METHOD METH_RecipeFileInit : BOOL
VAR_INPUT
END_VAR
aRecipeParamsVariables[0]  :=  'stUBL.nRecipeIndexShow.diValue := '																				;   
aRecipeParamsVariables[1]  :=  'stUBL.iPackageCapTypeShow.diValue := '																	;       
aRecipeParamsVariables[2]  :=  'stUBL.iPackageCapDiameterShow.diValue := '																	;       
aRecipeParamsVariables[3]  :=  'stUBL.bExEnableShow.bValue := '																			;        
aRecipeParamsVariables[4]  :=  'stUBL.bBottleFeederEnableShow.bValue := '																;     
aRecipeParamsVariables[5]  :=  'stUBL.iBottleFeederTurntableVelocitySVShow.diValue := '																;        
aRecipeParamsVariables[6]  :=  'stUBL.iBottleFeederBottleSensorDelayShow.diValue := '																	;             
aRecipeParamsVariables[7]  :=  'stUBL.iBottleFeederFormGateDelayShow.diValue := '																	;             
aRecipeParamsVariables[8]  :=  'stUBL.iBottleFeederAllowFormDelayShow.diValue := '																	;               
aRecipeParamsVariables[9]  :=  'stUBL.bPucksInserterEnableShow.bValue := '															;
aRecipeParamsVariables[10] := 'stUBL.iPucksInserterTurntableVelocitySVShow.diValue := '															;    
aRecipeParamsVariables[11] := 'stUBL.iPucksInserterConveyorVelocitySVShow.diValue := '															;		
aRecipeParamsVariables[12] := 'stUBL.iPucksInserterBottleSensorDelayShow.diValue := '															;	
aRecipeParamsVariables[13] := 'stUBL.iPucksInserterFormGateDelayShow.diValue := '														;	
aRecipeParamsVariables[14] := 'stUBL.iPucksInserterAllowFormDelayShow.diValue := '														;	
aRecipeParamsVariables[15] := 'stUBL.lrPucksInserterWheelOffsetShow.lrValue := '															;
aRecipeParamsVariables[16] := 'stUBL.lrPucksInserterWheelAccelerationShow.lrValue := '																;			
aRecipeParamsVariables[17] := 'stUBL.lrPucksInserterWheelVelocityShow.lrValue := '																;			
aRecipeParamsVariables[18] := 'stUBL.lrPucksInserterHammerHeightSVShow.lrValue := '																;			
aRecipeParamsVariables[19] := 'stUBL.bGateBeforeDispencersEnableShow.bValue := '																;			
aRecipeParamsVariables[20] := 'stUBL.nGateBeforeDispencersTimeFormInsertingShow.lrValue := '																;			
aRecipeParamsVariables[21] := 'stUBL.bGateAfterWeightEnableShow.bValue := '																;			
aRecipeParamsVariables[22] := 'stUBL.nGateAfterWeightTimeFormInsertingShow.lrValue := '															;
aRecipeParamsVariables[23] := 'stUBL.bGateRobotEnableShow.bValue := '		      																	  ;
aRecipeParamsVariables[24] := 'stUBL.nGateRobotTimeFormInsertingShow.lrValue := '															            ;
aRecipeParamsVariables[25] := 'stUBL.bFormsDragingLeftEnableShow.bValue := '	        												    ;
aRecipeParamsVariables[26] := 'stUBL.lrFormsDragingLeftVelocityShow.lrValue := '	        												    ;
aRecipeParamsVariables[27] := 'stUBL.lrFormsDragingLeftAccelerationShow.lrValue := '														   	        ;
aRecipeParamsVariables[28] := 'stUBL.lrFormsDragingLeftDecelerationShow.lrValue := '	   													            ;
aRecipeParamsVariables[29] := 'stUBL.bFormsDragingRightEnableShow.bValue := '															            ;
aRecipeParamsVariables[30] := 'stUBL.lrFormsDragingRightVelocityShow.lrValue := '															            ;
aRecipeParamsVariables[31] := 'stUBL.lrFormsDragingRightAccelerationShow.lrValue := '															            ;
aRecipeParamsVariables[32] := 'stUBL.lrFormsDragingRightDecelerationShow.lrValue := '															            ;
aRecipeParamsVariables[33] := 'stUBL.bDosingTwoPhasesShow.bValue := '			        												    ;
aRecipeParamsVariables[34] := 'stUBL.lrDispencersLifterReadyPositionShow.lrValue := '															            ;
aRecipeParamsVariables[35] := 'stUBL.uiDispencerStartDosingDelayShow.udiValue := '														        ;
aRecipeParamsVariables[36] := 'stUBL.bDispencer1EnableShow.bValue := '	          																									  ;
aRecipeParamsVariables[37] := 'stUBL.bDispencer2EnableShow.bValue := '			  																									      ;
aRecipeParamsVariables[38] := 'stUBL.bDispencer3EnableShow.bValue := '	          													  ;
aRecipeParamsVariables[39] := 'stUBL.bDispencer4EnableShow.bValue := '				       									     ;
aRecipeParamsVariables[40] := 'stUBL.lrDispencer1DoseVolumeShow.lrValue := '				   									         ;
aRecipeParamsVariables[41] := 'stUBL.lrDispencer1Phase1VolumeShow.lrValue:= '	           									             ;
aRecipeParamsVariables[42] := 'stUBL.lrDispencer1Phase2VolumeShow.lrValue := '		       									         ;
aRecipeParamsVariables[43] := 'stUBL.lrDispencer1Phase1VelocityShow.lrValue := '		       									         ;
aRecipeParamsVariables[44] := 'stUBL.lrDispencer1Phase2VelocityShow.lrValue := '															;
aRecipeParamsVariables[45] := 'stUBL.lrDispencer1Phase3VelocityShow.lrValue := '			   									             ;
aRecipeParamsVariables[46] := 'stUBL.lrDispencer1SuckVelocityShow.lrValue := '			   									             ;
aRecipeParamsVariables[47] := 'stUBL.lrDispencer1Phase1AccelerationShow.lrValue := '												                ;
aRecipeParamsVariables[48] := 'stUBL.lrDispencer1Phase2AccelerationShow.lrValue := '		   									             ;
aRecipeParamsVariables[49] := 'stUBL.lrDispencer1Phase3AccelerationShow.lrValue := '		   									             ;
aRecipeParamsVariables[50] := 'stUBL.lrDispencer1SuckAccelerationShow.lrValue := '		   									             ;
aRecipeParamsVariables[51] := 'stUBL.lrDispencer1Phase1DecelerationShow.lrValue := '	       									         ;
aRecipeParamsVariables[52] := 'stUBL.lrDispencer1Phase2DecelerationShow.lrValue := '												                ;
aRecipeParamsVariables[53] := 'stUBL.lrDispencer1Phase3DecelerationShow.lrValue := '		   									                 ;
aRecipeParamsVariables[54] := 'stUBL.udiDispencer1DosingDoneDelayTimeShow.udiValue := '											                    ;
aRecipeParamsVariables[55] := 'stUBL.lrDispencer1SuckValveOpenVolumeShow.lrValue := '											                ;
aRecipeParamsVariables[56] := 'stUBL.lrDispencer1SuckValveOpenTimeDelayShow.lrValue := '											                ;
aRecipeParamsVariables[57] := 'stUBL.lrDispencer1SuckValveCloseVolumeShow.lrValue := '											                ;
aRecipeParamsVariables[58] := 'stUBL.lrDispencer1SuckValveCloseTimeDelayShow.lrValue := '										                    ;
aRecipeParamsVariables[59] := 'stUBL.lrDispencer1DoseValveOpenVolumeShow.lrValue := '	   									             ;
aRecipeParamsVariables[60] := 'stUBL.lrDispencer1DoseValveOpenTimeAccShow.lrValue := '      									               ;
aRecipeParamsVariables[61] := 'stUBL.lrDispencer1DoseValveCloseVolumeShow.lrValue := '      									               ;
aRecipeParamsVariables[62] := 'stUBL.lrDispencer1DoseValveCloseTimeDecShow.lrValue := '												                ;
aRecipeParamsVariables[63] := 'stUBL.lrDispencer1DoseSuckingVolumeShow.lrValue := '												                ;
aRecipeParamsVariables[64] := 'stUBL.lrDispencer1DoseSuckingTimeDelayShow.lrValue := '												                ;
aRecipeParamsVariables[65] := 'stUBL.bDispencer1DoseSuckingShow.bValue := '			       									         ;
aRecipeParamsVariables[66] := 'stUBL.bDispencer1LiftSynchroPh1Show.bValue := '																;
aRecipeParamsVariables[67] := 'stUBL.bDispencer1LiftSynchroPh2Show.bValue := '			   									             ;
aRecipeParamsVariables[68] := 'stUBL.bDispencer1LiftSynchroPh3Show.bValue := '		       									         ;
aRecipeParamsVariables[69] := 'stUBL.lrDispencer1LifterStartDosePositionShow.lrValue := '								                ;
aRecipeParamsVariables[70] := 'stUBL.lrDispencer1LifterStopDosePositionShow.lrValue := '										                ;
aRecipeParamsVariables[71] := 'stUBL.lrDispencer1LifterVelocityShow.lrValue := '	            							    ;
aRecipeParamsVariables[72] := 'stUBL.lrDispencer1LifterAccelerationShow.lrValue := '	        							        ;
aRecipeParamsVariables[73] := 'stUBL.lrDispencer1LifterDecelerationShow.lrValue := '		    							            ;
aRecipeParamsVariables[74] := 'stUBL.lrDispencer2DoseVolumeShow.lrValue := '		            							    ;
aRecipeParamsVariables[75] := 'stUBL.lrDispencer2Phase1VolumeShow.lrValue := '			    							            ;
aRecipeParamsVariables[76] := 'stUBL.lrDispencer2Phase2VolumeShow.lrValue := '			    							            ;
aRecipeParamsVariables[77] := 'stUBL.lrDispencer2Phase1VelocityShow.lrValue := '			    							            ;
aRecipeParamsVariables[78] := 'stUBL.lrDispencer2Phase2VelocityShow.lrValue := '			    							            ;
aRecipeParamsVariables[79] := 'stUBL.lrDispencer2Phase3VelocityShow.lrValue := '			    							            ;
aRecipeParamsVariables[80] := 'stUBL.lrDispencer2SuckVelocityShow.lrValue := '			    							            ;
aRecipeParamsVariables[81] := 'stUBL.lrDispencer2Phase1AccelerationShow.lrValue := '	        							        ;
aRecipeParamsVariables[82] := 'stUBL.lrDispencer2Phase2AccelerationShow.lrValue := '	        							        ;
aRecipeParamsVariables[83] := 'stUBL.lrDispencer2Phase3AccelerationShow.lrValue := '		    							            ;
aRecipeParamsVariables[84] := 'stUBL.lrDispencer2SuckAccelerationShow.lrValue := '	        							        ;
aRecipeParamsVariables[85] := 'stUBL.lrDispencer2Phase1DecelerationShow.lrValue := '											                ;
aRecipeParamsVariables[86] := 'stUBL.lrDispencer2Phase2DecelerationShow.lrValue := '											                ;
aRecipeParamsVariables[87] := 'stUBL.lrDispencer2Phase3DecelerationShow.lrValue := '											                ;
aRecipeParamsVariables[88] := 'stUBL.udiDispencer2DosingDoneDelayTimeShow.udiValue := '													;
aRecipeParamsVariables[89] := 'stUBL.lrDispencer2SuckValveOpenVolumeShow.lrValue := '									                ;
aRecipeParamsVariables[90] := 'stUBL.lrDispencer2SuckValveOpenTimeDelayShow.lrValue := '											                ;
aRecipeParamsVariables[91] := 'stUBL.lrDispencer2SuckValveCloseVolumeShow.lrValue := '											                ;
aRecipeParamsVariables[92] := 'stUBL.lrDispencer2SuckValveCloseTimeDelayShow.lrValue := '											                ;
aRecipeParamsVariables[93] := 'stUBL.lrDispencer2DoseValveOpenVolumeShow.lrValue := '										                ;
aRecipeParamsVariables[94] := 'stUBL.lrDispencer2DoseValveOpenTimeAccShow.lrValue := '									                    ;
aRecipeParamsVariables[95] := 'stUBL.lrDispencer2DoseValveCloseVolumeShow.lrValue := '									                    ;
aRecipeParamsVariables[96] := 'stUBL.lrDispencer2DoseValveCloseTimeDecShow.lrValue := '										                    ;
aRecipeParamsVariables[97] := 'stUBL.lrDispencer2DoseSuckingVolumeShow.lrValue := '		    							                    ;
aRecipeParamsVariables[98] := 'stUBL.lrDispencer2DoseSuckingTimeDelayShow.lrValue := '									                        ;
aRecipeParamsVariables[99] := 'stUBL.bDispencer2DoseSuckingShow.bValue := '		            							        ;
aRecipeParamsVariables[100]:= 'stUBL.bDispencer2LiftSynchroPh1Show.bValue := '		        							            ;
aRecipeParamsVariables[101]:= 'stUBL.bDispencer2LiftSynchroPh2Show.bValue := '		        							            ;
aRecipeParamsVariables[102]:= 'stUBL.bDispencer2LiftSynchroPh3Show.bValue := '		        							        ;
aRecipeParamsVariables[103]:= 'stUBL.lrDispencer2LifterStartDosePositionShow.lrValue := '								  	                    ;
aRecipeParamsVariables[104]:= 'stUBL.lrDispencer2LifterStopDosePositionShow.lrValue := '								  	            ;
aRecipeParamsVariables[105]:= 'stUBL.lrDispencer2LifterVelocityShow.lrValue := '	        							            ;
aRecipeParamsVariables[106]:= 'stUBL.lrDispencer2LifterAccelerationShow.lrValue := '									                ;
aRecipeParamsVariables[107]:= 'stUBL.lrDispencer2LifterDecelerationShow.lrValue := '	    							                ;
aRecipeParamsVariables[108]:= 'stUBL.bDispencersCatchEnableShow.bValue := '	            							    ;
aRecipeParamsVariables[109]:= 'stUBL.bDispencersCatchMaxPressureShow.bValue := '           							         ;
aRecipeParamsVariables[110]:= 'stUBL.lrDispencersCatchHeightSVShow.lrValue := '														;
aRecipeParamsVariables[111]:= 'stUBL.lrDispencersCatch1ClosedValueShow.lrValue := '         							       ;
aRecipeParamsVariables[112]:= 'stUBL.lrDispencersCatch1OpenValueShow.lrValue := '           							   ;
aRecipeParamsVariables[113]:= 'stUBL.lrDispencersCatch2ClosedValueShow.lrValue := '         							         ;
aRecipeParamsVariables[114]:= 'stUBL.lrDispencersCatch2OpenValueShow.lrValue := '		    							            ;
aRecipeParamsVariables[115]:= 'stUBL.lrDispencersCatch3ClosedValueShow.lrValue := '         							       ;
aRecipeParamsVariables[116]:= 'stUBL.lrDispencersCatch3OpenValueShow.lrValue := '           							        ;
aRecipeParamsVariables[117]:= 'stUBL.lrDispencersCatch4ClosedValueShow.lrValue := '         							        ;
aRecipeParamsVariables[118]:= 'stUBL.lrDispencersCatch4OpenValueShow.lrValue := '										;								
aRecipeParamsVariables[119]:= 'stUBL.lrDispencersCatchToleranceShow.lrValue := '	        							;
aRecipeParamsVariables[120]:= 'stUBL.bTank1MixerEnableShow.bValue := '    												 ;
aRecipeParamsVariables[121]:= 'stUBL.bTankHeatingEnableShow.bValue := '   												                ;
aRecipeParamsVariables[122]:= 'stUBL.iTankHeatingTempSVShow.diValue := '   												      ;
aRecipeParamsVariables[123]:= 'stUBL.bTank1PressureEnableShow.bValue := ' 														;
aRecipeParamsVariables[124]:= 'stUBL.bTank1SupplyPumpEnableShow.bValue := '	                                           ;
aRecipeParamsVariables[125]:= 'stUBL.bTank2SupplyPumpEnableShow.bValue := '	                                           ;
aRecipeParamsVariables[126]:= 'stUBL.uTank1LevelSetpointShow.udiValue := '	                                           ;
aRecipeParamsVariables[127]:= 'stUBL.uTank2LevelSetpointShow.udiValue := '	                                           ;
aRecipeParamsVariables[128]:= 'stUBL.bTank1LevelSignalInvertShow.bValue := '	                                           ;
aRecipeParamsVariables[129]:= 'stUBL.bTank2LevelSignalInvertShow.bValue := '	                                           ;
aRecipeParamsVariables[130]:= 'stUBL.bWeight1EnableShow.bValue := '	                                           ;
aRecipeParamsVariables[131]:= 'stUBL.lrWeightMassSVShow.lrValue := '	                                           ;
aRecipeParamsVariables[132]:= 'stUBL.iWeight1ActuatorUpDelayShow.diValue := '											  ;	
aRecipeParamsVariables[133]:= 'stUBL.iWeight2ActuatorUpDelayShow.diValue := '	                                           ;
aRecipeParamsVariables[134]:= 'stUBL.iWeight3ActuatorUpDelayShow.diValue := '	                                           ;
aRecipeParamsVariables[135]:= 'stUBL.iWeight4ActuatorUpDelayShow.diValue := '	                                           ;
aRecipeParamsVariables[136]:= 'stUBL.iWeight5ActuatorUpDelayShow.diValue := '	                                           ;
aRecipeParamsVariables[137]:= 'stUBL.iWeight6ActuatorUpDelayShow.diValue := '	                                           ;
aRecipeParamsVariables[138]:= 'stUBL.lrFormWeightShow.lrValue := '	                                           ;
aRecipeParamsVariables[139]:= 'stUBL.lrMass1DensityShow.lrValue := '	                                           ;
aRecipeParamsVariables[140]:= 'stUBL.lrMass2DensityShow.lrValue := '	                                           ;
aRecipeParamsVariables[141]:= 'stUBL.lrCupWeightShow.lrValue := '	                                           ;
aRecipeParamsVariables[142]:= 'stUBL.lrWholePackageWeightShow.lrValue := '	                                           ;
aRecipeParamsVariables[143]:= 'stUBL.lrWeight1MeasurmentCorrectionShow.lrValue := '	                                           ;
aRecipeParamsVariables[144]:= 'stUBL.bDispencer1WeightCorrectionEnableShow.bValue := '	                                           ;
aRecipeParamsVariables[145]:= 'stUBL.bDispencer2WeightCorrectionEnableShow.bValue := '	                                           ;
aRecipeParamsVariables[146]:= 'stUBL.bDispencer3WeightCorrectionEnableShow.bValue := '	                                           ;
aRecipeParamsVariables[147]:= 'stUBL.bDispencer4WeightCorrectionEnableShow.bValue := '	                                           ;
aRecipeParamsVariables[148]:= 'stUBL.lrWeightUpperToleranceShow.lrValue := '	                                           ;
aRecipeParamsVariables[149]:= 'stUBL.lrWeightLowerToleranceShow.lrValue := '	                                           ;
aRecipeParamsVariables[150]:= 'stUBL.iWeightCorrectionNumberOfSamplesShow.diValue := '	                                           ;
aRecipeParamsVariables[151]:= 'stUBL.bLidFeederEnableShow.bValue := '	                                           ;
aRecipeParamsVariables[152]:= 'stUBL.bLidFeederHeaterEnableShow.bValue := '	                                           ;
aRecipeParamsVariables[153]:= 'stUBL.lrLidFeederHeightPosSVShow.lrValue := '	                                           ;
aRecipeParamsVariables[154]:= 'stUBL.iLidFeederHeatingTimeShow.diValue := '	                                           ;
aRecipeParamsVariables[155]:= 'stUBL.iLidFeederTempHisteresisShow.diValue := '	                                           ;
aRecipeParamsVariables[156]:= 'stUBL.iLidFeeder1TempSVShow.diValue := '	                                           ;
aRecipeParamsVariables[157]:= 'stUBL.iLidFeeder2TempSVShow.diValue := '	                                           ;
aRecipeParamsVariables[158]:= 'stUBL.bLidFeederDragingStationEnableShow.bValue := '	                                           ;
aRecipeParamsVariables[159]:= 'stUBL.lrLidFeederDragingStationVelocityShow.lrValue := '	                                           ;
aRecipeParamsVariables[160]:= 'stUBL.lrLidFeederDragingStationAccelerationShow.lrValue := '	                                           ;
aRecipeParamsVariables[161]:= 'stUBL.lrLidFeederDragingStationDecelerationShow.lrValue := '	                                           ;
aRecipeParamsVariables[162]:= 'stUBL.bLidPuttedCheckEnableShow.bValue := '	                                           ;
aRecipeParamsVariables[163]:= 'stUBL.lrLidPuttedCheckHeightSVShow.lrValue := '	                                           ;
aRecipeParamsVariables[164]:= 'stUBL.lrLidPuttedCheckPositionShow.lrValue := '	                                           ;
aRecipeParamsVariables[165]:= 'stUBL.lrLidPuttedCheckAreaShow.lrValue := '	                                           ;
aRecipeParamsVariables[166]:= 'stUBL.iLidPuttedCheckProgramShow.diValue := '	                                           ;
aRecipeParamsVariables[167]:= 'stUBL.bLidSealerEnableSho.bValuew := '	                                           ;
aRecipeParamsVariables[168]:= 'stUBL.bLidSealerHeaterEnableShow.bValue := '	                                           ;
aRecipeParamsVariables[169]:= 'stUBL.iLidSealerHeatingTimeShow.diValue := '	                                           ;
aRecipeParamsVariables[170]:= 'stUBL.lrLidSealerPressureShow.lrValue := '	                                           ;
aRecipeParamsVariables[171]:= 'stUBL.lrLidSealerHeightPosSVShow.lrValue := '	                                           ;
aRecipeParamsVariables[172]:= 'stUBL.iLidSealerTempHisteresisShow.diValue := '	                                           ;
aRecipeParamsVariables[173]:= 'stUBL.iLidSealer1TempSVShow.diValue := '	                                           ;
aRecipeParamsVariables[174]:= 'stUBL.iLidSealer2TempSVShow.diValue := '	                                           ;
aRecipeParamsVariables[175]:= 'stUBL.bLidSealerDragingStationEnableShow.bValue := '	                                           ;
aRecipeParamsVariables[176]:= 'stUBL.lrLidSealerDragingStationVelocityShow.lrValue := '	                                           ;
aRecipeParamsVariables[177]:= 'stUBL.lrLidSealerDragingStationAccelerationShow.lrValue := '	                                           ;
aRecipeParamsVariables[178]:= 'stUBL.lrLidSealerDragingStationDecelerationShow.lrValue := '	                                           ;
aRecipeParamsVariables[179]:= 'stUBL.bCapFeederGateEnableShow.bValue := '	                                           ;
aRecipeParamsVariables[180]:= 'stUBL.iCapFeederGateBlockingTimeShow.diValue := '	                                           ;
aRecipeParamsVariables[181]:= 'stUBL.bCapFeederEnableShow.bValue := '	                                           ;
aRecipeParamsVariables[182]:= 'stUBL.lrCapFeederHeightPosSVShow.lrValue := '	                                           ;
aRecipeParamsVariables[183]:= 'stUBL.iCapFeederTimeDelayOnShow.diValue := '                                            ;
aRecipeParamsVariables[184]:= 'stUBL.iCapFeederTimeDelayOffShow.diValue := '                                            ;
aRecipeParamsVariables[185]:= 'stUBL.iCapFeederTimeToEmptySleeveErrorShow.diValue := '	                                           ;
aRecipeParamsVariables[186]:= 'stUBL.bCapSorterOnlyWeightOKEnableShow.bValue := '	                                           ;
aRecipeParamsVariables[187]:= 'stUBL.bCapSorterDragEnableShow.bValue := '	                                           ;
aRecipeParamsVariables[188]:= 'stUBL.lrCapSorterDragVelocityShow.lrValue := '	                                           ;
aRecipeParamsVariables[189]:= 'stUBL.lrCapSorterDragAccelerationShow.lrValue := '	                                           ;
aRecipeParamsVariables[190]:= 'stUBL.lrCapSorterDragDecelerationShow.lrValue := '	                                           ;
aRecipeParamsVariables[191]:= 'stUBL.bCapPuttedCheckEnableShow.bValue := '	                                           ;
aRecipeParamsVariables[192]:= 'stUBL.lrCapPuttedCheckHeightPosSVShow.lrValue := '	                                           ;
aRecipeParamsVariables[193]:= 'stUBL.bGripperScrewer1EnableShow.bValue := '	                                           ;
aRecipeParamsVariables[194]:= 'stUBL.lrGripperScrewingTightTorqueShow.lrValue := '	                                           ;
aRecipeParamsVariables[195]:= 'stUBL.bGripperScrewer2EnableShow.bValue := '	                                           ;
aRecipeParamsVariables[196]:= 'stUBL.lrGripperScrewing2TightTorqueShow.lrValue := '	                                           ;
aRecipeParamsVariables[197]:= 'stUBL.iGripperScrewer1ToolShow.diValue := '	                                           ;
aRecipeParamsVariables[198]:= 'stUBL.lrGripperScrewer1VelocityShow.lrValue := '	                                           ;
aRecipeParamsVariables[199]:= 'stUBL.nGripperScrewer1TightTimeShow.udiValue := '	                                           ;
aRecipeParamsVariables[200]:= 'stUBL.iGripperScrewer1StartDelayShow.diValue := '	                                           ;
aRecipeParamsVariables[201]:= 'stUBL.lrGripperScrewerReadyPositionShow.lrValue := '	                                           ;
aRecipeParamsVariables[202]:= 'stUBL.lrGripperScrewerPushingCapPositionShow.lrValue := '	                                           ;
aRecipeParamsVariables[203]:= 'stUBL.lrGripperScrewerScrewingCapPositionShow.lrValue := '	                                           ;
aRecipeParamsVariables[204]:= 'stUBL.lrGripperScrewerPressureShow.lrValue := '	                                           ;
aRecipeParamsVariables[205]:= 'stUBL.lrGripperScrewerCatchPressureShow.lrValue := '	                                           ;
aRecipeParamsVariables[206]:= 'stUBL.lrDispencerCatchPressureShow.lrValue := '	                                           ;
aRecipeParamsVariables[207]:= 'stUBL.lrGripperScrewerPressureExhaustLevelShow.lrValue := '	                                           ;
aRecipeParamsVariables[208]:= 'stUBL.lrGripperScrewerCatchPressureExhaustLevelShow.lrValue := '	                                           ;
aRecipeParamsVariables[209]:= 'stUBL.lrGripperScrewerTurnoversToFullScrewedShow.lrValue := '	                                           ;
aRecipeParamsVariables[210]:= 'stUBL.lrGripperScrewerThreadPitchShow.lrValue := '	                                           ;
aRecipeParamsVariables[211]:= 'stUBL.lrGripperScrewerThreadTimesShow.lrValue := '	                                           ;
aRecipeParamsVariables[212]:= 'stUBL.nGripperScrewerCatchHeightSVShow.udiValue := '	                           								                ;
aRecipeParamsVariables[213]:= 'stUBL.bGripperScrewer1FindScrewShow.bValue := '	                		            ;
aRecipeParamsVariables[214]:= 'stUBL.bGripperScrewer1Option4Show.bValue := '	                		            ;
aRecipeParamsVariables[215]:= 'stUBL.lrGripperScrewer1FindingScrewDegreeShow.lrValue := '	    		                        ;
aRecipeParamsVariables[216]:= 'stUBL.bGripperScrewer1Option1Show.bValue := '	                		            ;
aRecipeParamsVariables[217]:= 'stUBL.bGripperScrewer1Option2Show.bValue := '	                		            ;
aRecipeParamsVariables[218]:= 'stUBL.bGripperScrewer1Option3Show.bValue := '	                		            ;
aRecipeParamsVariables[219]:= 'stUBL.bGripperScrewer1Option5Show.bValue := '	                		            ;
aRecipeParamsVariables[220]:= 'stUBL.bGripperScrewer1Option6Show.bValue := '	                		            ;
aRecipeParamsVariables[221]:= 'stUBL.bGripperScrewer1Option7Show.bValue := '	                		            ;
aRecipeParamsVariables[222]:= 'stUBL.bBottleDragingStationEnableShow.bValue := '	            		                ;
aRecipeParamsVariables[223]:= 'stUBL.lrBottleDragingStationVelocityShow.lrValue := '	        		                    ;
aRecipeParamsVariables[224]:= 'stUBL.bCapCorrectCheckEnableShow.bValue := '	                    	            ;
aRecipeParamsVariables[225]:= 'stUBL.lrCapCorrectCheckHeightPosSVShow.lrValue := '	            		                ;
aRecipeParamsVariables[226]:= 'stUBL.bCapCorrectCheckCameraEnableShow.bValue := '	            		                ;
aRecipeParamsVariables[227]:= 'stUBL.iCapCorrectCheckCameraProgramShow.diValue := '	            		                ;
aRecipeParamsVariables[228]:= 'stUBL.bBottleTransferEnableShow.bValue		 := '	            		                ;
aRecipeParamsVariables[229]:= 'stUBL.nBottleTransferProgramShow.udiValue		 := '	        			                ;
aRecipeParamsVariables[230]:= 'stUBL.iBottleTransferPickOffsetXShow.diValue  := '	            		                ;
aRecipeParamsVariables[231]:= 'stUBL.iBottleTransferPickOffsetYShow.diValue  := '	            		                ;
aRecipeParamsVariables[232]:= 'stUBL.iBottleTransferPickOffsetZShow.diValue  := '	            		                ;
aRecipeParamsVariables[233]:= 'stUBL.iBottleTransferPick2OffsetXShow.diValue := '	            		                ;
aRecipeParamsVariables[234]:= 'stUBL.iBottleTransferPick2OffsetYShow.diValue := '	            		                ;
aRecipeParamsVariables[235]:= 'stUBL.iBottleTransferPick2OffsetZShow.diValue := '	            		                ;
aRecipeParamsVariables[236]:= 'stUBL.iBottleTransferPlace1OffsetXShow.diValue := '	            		                ;
aRecipeParamsVariables[237]:= 'stUBL.iBottleTransferPlace1OffsetYShow.diValue := '	            		                ;
aRecipeParamsVariables[238]:= 'stUBL.iBottleTransferPlace1OffsetZShow.diValue := '	            		                ;
aRecipeParamsVariables[239]:= 'stUBL.iBottleTransferPlace2OffsetXShow.diValue := '	            		                ;
aRecipeParamsVariables[240]:= 'stUBL.iBottleTransferPlace2OffsetYShow.diValue := '	            		                ;
aRecipeParamsVariables[241]:= 'stUBL.iBottleTransferPlace2OffsetZShow.diValue := '	            		                ;
aRecipeParamsVariables[242]:= 'stUBL.iBottleTransferSpeedShow.diValue := '	                    		        ;
aRecipeParamsVariables[243]:= 'stUBL.bBottleTransferInkJetEnableShow.bValue := '	            		                ;
aRecipeParamsVariables[244]:= 'stUBL.bBottleTransferPickOnlyOneShow.bValue := '	                	                ;
aRecipeParamsVariables[245]:= 'stUBL.bBottleTransferWeightEnableShow.bValue := '	            		  							              ;
aRecipeParamsVariables[246]:= 'stUBL.iBottleTransferWeightIntervalShow.diValue := '	            		              ;
aRecipeParamsVariables[247]:= 'stUBL.bBottleTransferRotateEnableShow.bValue := '	            		              ;
aRecipeParamsVariables[248]:= 'stUBL.bBadBottleConveyorEnableShow.bValue := '	                		          ;
aRecipeParamsVariables[249]:= 'stUBL.nBadBottleConveyorVelocitySVShow.udiValue := '	            		              ;
aRecipeParamsVariables[250]:= 'stUBL.bLabelMachineEnableShow.bValue := '	                    		      ;
aRecipeParamsVariables[251]:= 'stUBL.bExitTurnTable1EnableShow.bValue := '	                    		      ;
aRecipeParamsVariables[252]:= 'stUBL.bExitConveyorEnableShow.bValue := '	                    		      ;
aRecipeParamsVariables[253]:= 'stUBL.nExitConveyorVelocitySVShow.udiValue := '	                		          ;
aRecipeParamsVariables[254]:= 'stUBL.bFormTransportersEnableShow.bValue					 := '		                              ;
aRecipeParamsVariables[255]:= 'stUBL.nFormTransportersDispencerVelocitySVShow.udiValue	 := '	                 							                          ;
aRecipeParamsVariables[256]:= 'stUBL.nFormTransportersScrewerVelocitySVShow.udiValue		 := '	                 							                          ;
aRecipeParamsVariables[257]:= 'stUBL.nFormTransportersBeforeScrewerVelocitySVShow.udiValue := '	                 				                          ;
aRecipeParamsVariables[258]:= 'stUBL.nFormTransportersSlowerVelocitySVShow.udiValue		 := '	                 				                          ;
aRecipeParamsVariables[259]:= 'stUBL.bCircularInkjetEnableShow.bValue	 := '	                                 				          ;
aRecipeParamsVariables[260]:= 'stUBL.iCircularInkjetSpeedShow.diValue	 := '	                                 				          ;
aRecipeParamsVariables[261]:= 'stUBL.iCircularInkjetDelayShow.diValue	 := '	                                 				          ;
aRecipeParamsVariables[262]:= 'stUBL.iCircularInkjetHoldShow.diValue	 := '	                                 				          ;
aRecipeParamsVariables[263]:= 'stUCF.iCapSorterProductType.diValue := '	                                         								  ;
aRecipeParamsVariables[264]:= 'stUCF.uiCapSorterIndexShow.udiValue := '																						;
aRecipeParamsVariables[265]:= 'stUCF.bPresenceBottleEnableShow.bValue := '	                                     									                                ;
aRecipeParamsVariables[266]:= 'stUCF.bCapSorterTransporterEnableShow.bValue								 := '	  					     ;
aRecipeParamsVariables[267]:= 'stUCF.iCapSorterTransporterTankConveyorVelocityShow.diValue				 := '	    					   ;
aRecipeParamsVariables[268]:= 'stUCF.iCapSorterTransporterStartDelayTimeShow.diValue						 := '						  ;
aRecipeParamsVariables[269]:= 'stUCF.udiCapSorterTransporterTimeProductOnSensorBeforeBrushShow.udiValue	 := '										            ;
aRecipeParamsVariables[270]:= 'stUCF.iCapSorterTransporterEmptyingConveyorSpeedShow.diValue				 := '					            ;
aRecipeParamsVariables[271]:= 'stUCF.iCapSorterTransporterVolumeOfCapsShow.diValue						 := '					            ;
aRecipeParamsVariables[272]:= 'stUCF.bCapSorterWheelEnableShow.bValue							 := '	        				     ;
aRecipeParamsVariables[273]:= 'stUCF.lrCapSorterWheelMoveAccelerationEmptyTableShow.lrValue		 := '	        				   	 ;
aRecipeParamsVariables[274]:= 'stUCF.lrCapSorterWheelMoveDecelerationEmptyTableShow.lrValue		 := '	        				   	 ;
aRecipeParamsVariables[275]:= 'stUCF.lrCapSorterWheelMoveSpeedEmptyTableShow.lrValue				 := '	    				        ;
aRecipeParamsVariables[276]:= 'stUCF.lrCapSorterWheelMoveAngleEmptyTableShow.lrValue				 := '	    				        ;
aRecipeParamsVariables[277]:= 'stUCF.lrCapSorterWheelJerkAngleEmptyTableShow.lrValue				 := '	    				        ;
aRecipeParamsVariables[278]:= 'stUCF.iCapSorterWheelWaitingAfterRotationEmptyTableShow.diValue := '	            				    ;
aRecipeParamsVariables[279]:= 'stUCF.lrCapSorterWheelMoveAccelerationFullTableShow.lrValue	 := '	            				    ;
aRecipeParamsVariables[280]:= 'stUCF.lrCapSorterWheelMoveDecelerationFullTableShow.lrValue	 := '	            				   ;
aRecipeParamsVariables[281]:= 'stUCF.lrCapSorterWheelMoveSpeedFullTableShow.lrValue			 := '	            				    ;
aRecipeParamsVariables[282]:= 'stUCF.lrCapSorterWheelMoveAngleFullyTableShow.lrValue			 := '           				   ;
aRecipeParamsVariables[283]:= 'stUCF.lrCapSorterWheelJerkAngleFullTableShow.lrValue			 := '               				   ;
aRecipeParamsVariables[284]:= 'stUCF.iCapSorterWheelWaitingAfterRotationFullTableShow.diValue := '	           											    ;
aRecipeParamsVariables[285]:= 'stUCF.lrCapSorterWheelMoveAccelerationHalfFullTableShow.lrValue	 := '	       											     ;
aRecipeParamsVariables[286]:= 'stUCF.lrCapSorterWheelMoveDecelerationHalfFullTableShow.lrValue	 := '	       				     ;
aRecipeParamsVariables[287]:= 'stUCF.lrCapSorterWheelMoveSpeedHalfFullTableShow.lrValue			 := '	       				     ;
aRecipeParamsVariables[288]:= 'stUCF.lrCapSorterWheelMoveAngleHalfFullyTableShow.lrValue			 := '	   				         ;
aRecipeParamsVariables[289]:= 'stUCF.lrCapSorterWheelJerkAngleHalfFullTableShow.lrValue			 := '	       				     ;
aRecipeParamsVariables[290]:= 'stUCF.iCapSorterWheelWaitingAfterRotationHalfFullTableShow.diValue := '	       				     ;
aRecipeParamsVariables[291]:= 'stUCF.bCapSorterCameraEnableShow.bValue := '     ;                             				
aRecipeParamsVariables[292]:= 'stUCF.bCapSorterRobotEnableShow.bValue := '	 ;                                 				
aRecipeParamsVariables[293]:= 'stUCF.lrCapSorterRobotPlace1PositionXShow.lrValue			 := '									     ;
aRecipeParamsVariables[294]:= 'stUCF.lrCapSorterRobotPlace1PositionYShow.lrValue			 := '									     ;
aRecipeParamsVariables[295]:= 'stUCF.lrCapSorterRobotPlace1PositionZShow.lrValue			 := '									     ;
aRecipeParamsVariables[296]:= 'stUCF.lrCapSorterRobotPlace1PositionCShow.lrValue			 := '									     ;
aRecipeParamsVariables[297]:= 'stUCF.iCapSorterRobotPickElevationShow.diValue			 := '	    								 ;
aRecipeParamsVariables[298]:= 'stUCF.iCapSorterRobotPickTimeShow.diValue					 := '									     ;
aRecipeParamsVariables[299]:= 'stUCF.iCapSorterRobotVacuumActivationShow.diValue			 := '									     ;
aRecipeParamsVariables[300]:= 'stUCF.iCapSorterRobotVacuumOffShow.diValue				 := '	    								 ;
aRecipeParamsVariables[301]:= 'stUCF.iCapSorterRobotPlaceTimeShow.diValue				 := '	    								 ;
aRecipeParamsVariables[302]:= 'stUCF.iCapSorterRobotTCP_PlaceOffsetShow.diValue			 := '	    								 ;
aRecipeParamsVariables[303]:= 'stUCF.iCapSorterRobotAccelerationDecelerationShow.diValue	 := '									     ;
aRecipeParamsVariables[304]:= 'stUCF.iCapSorterRobotGripperWatchdogShow.diValue			 := '	    								 ;
aRecipeParamsVariables[305]:= 'stUCF.iCapSorterRobotParalaxCorrectionShow.diValue		 := '	    								 ;
aRecipeParamsVariables[306]:= 'stUCF.iCapSorterRobotNumberToolShow.diValue	 := '	 													 ;
aRecipeParamsVariables[307]:= 'stUCF.iCapSorterRobotPickPositionZShow.diValue := '	 													 ;
aRecipeParamsVariables[308]:= 'stUCF.iCapSorterRobotTCP_Lenght.diValue		 := '	 																			 ;
aRecipeParamsVariables[309]:= 'stUCF.iCapSorterRobotProductDiametr.diValue	 := '	 												 ;
aRecipeParamsVariables[310]:= 'stUCF.bCapSorterIntermediateTransporterEnableShow.bValue					 := '				     ;
aRecipeParamsVariables[311]:= 'stUCF.iCapSorterIntermediateTransporterAutoSpeedShow.diValue				 := '	    			 ;
aRecipeParamsVariables[312]:= 'stUCF.iCapSorterIntermediateTransporterManualSpeedShow.diValue			 := '	    			 ;
aRecipeParamsVariables[313]:= 'stUCF.iCapSorterIntermediateTransporterEmptyingSpeedShow.diValue			 := '	    			 ;
aRecipeParamsVariables[314]:= 'stUCF.iCapSorterIntermediateTransporterDelayCountTimeShow.diValue			 := '				     ;
aRecipeParamsVariables[315]:= 'stUCF.iCapSorterIntermediateTransporterReverseTimeShow.diValue			 := '	    			 ;
aRecipeParamsVariables[316]:= 'stUCF.udiCapSorterIntermediateTransporterTimeProductOnSensorShow.udiValue	 := '					 ;
aRecipeParamsVariables[317]:= 'stUCF.lrCapSorterIntermediateTransporterWheelAngleShow.lrValue			 := '	    			 ;
aRecipeParamsVariables[318]:= 'stUCF.bCapSorterIntermediateBrushEnableShow.bValue			 := '	  												      ;
aRecipeParamsVariables[319]:= 'stUCF.iCapSorterIntermediateBrushAutoSpeedShow.diValue		 := '	  												      ;
aRecipeParamsVariables[320]:= 'stUCF.iCapSorterIntermediateBrushManualSpeedShow.diValue		 := '	  						      ;
aRecipeParamsVariables[321]:= 'stUCF.iCapSorterIntermediateBrushEmptyingSpeedShow.diValue	 := '	  						      ;
aRecipeParamsVariables[322]:= 'stUCF.lrCapSorterIntermediateBrushPositionHeightSVShow.lrValue := '    						    ;
aRecipeParamsVariables[323]:= 'stUCF.bCapSorterBrush1OnWheelEnableShow.bValue			 := '      														  ;
aRecipeParamsVariables[324]:= 'stUCF.iCapSorterBrush1OnWheelAutoSpeedShow.diValue		 := '      					  ;
aRecipeParamsVariables[325]:= 'stUCF.iCapSorterBrush1OnWheelManualSpeedShow.diValue		 := '      					  ;
aRecipeParamsVariables[326]:= 'stUCF.iCapSorterBrush1OnWheelEmptyingSpeedShow.diValue	 := '      					  ;
aRecipeParamsVariables[327]:= 'stUCF.lrCapSorterBrush1OnWheelPositionHeightSVShow.lrValue := '     					   ;
aRecipeParamsVariables[328]:= 'stUCF.bCapSorterBrush2OnWheelEnableShow.bValue			 := '      					  ;
aRecipeParamsVariables[329]:= 'stUCF.iCapSorterBrush2OnWheelAutoSpeedShow.diValue		 := '      					  ;
aRecipeParamsVariables[330]:= 'stUCF.iCapSorterBrush2OnWheelManualSpeedShow.diValue		 := '      					  ;
aRecipeParamsVariables[331]:= 'stUCF.iCapSorterBrush2OnWheelEmptyingSpeedShow.diValue	 := '      					  ;
aRecipeParamsVariables[332]:= 'stUCF.lrCapSorterBrush2OnWheelPositionHeightSVShow.lrValue := '     					   ;
aRecipeParamsVariables[333]:= 'stUCF.bCapSorterFeederEnableShow.bValue					 := '      					  ;
aRecipeParamsVariables[334]:= 'stUCF.bCapSorterFeederEnableTubeError.bValue				 := '  						  ;
aRecipeParamsVariables[335]:= 'stUCF.lrCapSorterFeederMover1InputPositionShow.lrValue	 := '      					  ;
aRecipeParamsVariables[336]:= 'stUCF.lrCapSorterFeederMover2InputPositionShow.lrValue	 := '      					  ;
aRecipeParamsVariables[337]:= 'stUCF.lrCapSorterFeederMover1OutputPositionShow.lrValue	 := '      					  ;
aRecipeParamsVariables[338]:= 'stUCF.lrCapSorterFeederMover2OutputPositionShow.lrValue	 := '      					  ;
aRecipeParamsVariables[339]:= 'stUCF.lrCapSorterFeederSlotDistanceShow.lrValue			 := '      					  ;
aRecipeParamsVariables[340]:= 'stUCF.lrCapSorterFeederMoverSpeedShow.lrValue				 := '  					      ;
aRecipeParamsVariables[341]:= 'stUCF.lrCapSorterFeederMoverAccelerationShow.lrValue		 := '      					  ;
aRecipeParamsVariables[342]:= 'stUCF.lrCapSorterFeederMoveJerkShow.lrValue				 := '      					  ;
aRecipeParamsVariables[343]:= 'stUCF.bCapSorterPreScrewerEnableShow.bValue			 := '          					    ;
aRecipeParamsVariables[344]:= 'stUCF.bCapSorterPreScrewerPicker1EnableShow.bValue := '            					  ;
aRecipeParamsVariables[345]:= 'stUCF.bCapSorterPreScrewerPicker2EnableShow.bValue := '            					  ;
aRecipeParamsVariables[346]:= 'stUCF.bCapSorterPreScrewerPicker3EnableShow.bValue := '           													   ;
aRecipeParamsVariables[347]:= 'stUCF.bCapSorterPreScrewerPicker4EnableShow.bValue := '           																   ;
aRecipeParamsVariables[348]:= 'stUCF.lrCapSorterPreScrewerPickZPositionShow.lrValue					 := '       																 ;
aRecipeParamsVariables[349]:= 'stUCF.lrCapSorterPreScrewerCatcherReleseShow.lrValue					 := '       																 ;
aRecipeParamsVariables[350]:= 'stUCF.lrCapSorterPreScrewerCapCatcherZPositionShow.lrValue			 := '       																 ;
aRecipeParamsVariables[351]:= 'stUCF.lrCapSorterPreScrewerTopZPositionShow.lrValue					 := '       																 ;
aRecipeParamsVariables[352]:= 'stUCF.lrCapSorterPreScrewerCartesianCatchZPositionShow.lrValue		 := '       																 ;
aRecipeParamsVariables[353]:= 'stUCF.lrCapSorterPreScrewerStrawCatcherZPositionShow.lrValue			 := '       																 ;
aRecipeParamsVariables[354]:= 'stUCF.LrCapSorterPreScrewerCheckStrawCatcherActuatorZPosition.lrValue	 := '   																     ;
aRecipeParamsVariables[355]:= 'stUCF.lrCapSorterPreScrewerScrewerStartZPositionShow.lrValue			 := '       																 ;
aRecipeParamsVariables[356]:= 'stUCF.lrCapSorterPreScrewerGripperOpenPositionShow.lrValue			 := '       																 ;
aRecipeParamsVariables[357]:= 'stUCF.lrCapSorterPreScrewerPlaceZPositionShow.lrValue					 := '   																     ;
aRecipeParamsVariables[358]:= 'stUCF.lrCapSorterPreScrewerBendingDistanceShow.lrValue := '            ;
aRecipeParamsVariables[359]:= 'stUCF.lrCapSorterPreScrewerStrawInsertDistance.lrValue := '            ;
aRecipeParamsVariables[360]:= 'stUCF.lrCapSorterPreScrewerPickXMover1PositionShow.lrValue := '            ;
aRecipeParamsVariables[361]:= 'stUCF.lrCapSorterPreScrewerPickXMover2PositionShow.lrValue := '            ;
aRecipeParamsVariables[362]:= 'stUCF.lrCapSorterPreScrewerPlaceXPositionShow.lrValue		 := '            ;
aRecipeParamsVariables[363]:= 'stUCF.lrCapSorterPreScrewerScrewFindingShow.lrValue	 := '            ;
aRecipeParamsVariables[364]:= 'stUCF.lrCapSorterPreScrewerScrewDistanceShow.lrValue := '            ;
aRecipeParamsVariables[365]:= 'stUCF.lrCapSorterPreScrewerPickerSpeedShow.lrValue		 := '            ;
aRecipeParamsVariables[366]:= 'stUCF.lrCapSorterPreScrewerPickerAccelerationShow.lrValue	 := '        ;
aRecipeParamsVariables[367]:= 'stUCF.lrCapSorterPreScrewerPickerJerkShow.lrValue			 := '        ;
aRecipeParamsVariables[368]:= 'stUCF.lrCapSorterPreScrewerCatcherSpeedShow.lrValue		 := '        ;
aRecipeParamsVariables[369]:= 'stUCF.lrCapSorterPreScrewerCatcherAccelerationShow.lrValue := '        ;
aRecipeParamsVariables[370]:= 'stUCF.lrCapSorterPreScrewerCatcherJerkShow.lrValue		 := '        ;
aRecipeParamsVariables[371]:= 'stUCF.lrCapSorterPreScrewerScrewSpeedShow.lrValue			 := '        ;
aRecipeParamsVariables[372]:= 'stUCF.lrCapSorterPreScrewerScrewAccelerationShow.lrValue	 := '        ;
aRecipeParamsVariables[373]:= 'stUCF.lrCapSorterPreScrewerScrewJerkShow.lrValue			 := '        ;
aRecipeParamsVariables[374]:= 'stUCF.lrCapSorterPreScrewerCatcherCatchingPositionShow.lrValue := '        ;
aRecipeParamsVariables[375]:= 'stUCF.lrCapSorterPreScrewerCatcherPlacePositionShow.lrValue	 := '        ;
aRecipeParamsVariables[376]:= 'stUCF.lrCapSorterPreScrewerCatcherHightSVShow.lrValue			 := '        ;
aRecipeParamsVariables[377]:= 'stUCF.bCapSorterPreScrewerBottleCatcherEnableShow.bValue		 := '        ;
aRecipeParamsVariables[378]:= 'stUCF.lrCapSorterPreScrewerBottleCatch1OpenValueShow.lrValue	 := '        ;
aRecipeParamsVariables[379]:= 'stUCF.lrCapSorterPreScrewerBottleCatch1CloseValueShow.lrValue	 := '        ;
aRecipeParamsVariables[380]:= 'stUCF.lrCapSorterPreScrewerBottleCatch2OpenValueShow.lrValue	 := '        ;
aRecipeParamsVariables[381]:= 'stUCF.lrCapSorterPreScrewerBottleCatch2CloseValueShow.lrValue	 := '        ;
aRecipeParamsVariables[382]:= 'stUCF.lrCapSorterPreScrewerBottleCatch3OpenValueShow.lrValue	 := '        ;
aRecipeParamsVariables[383]:= 'stUCF.lrCapSorterPreScrewerBottleCatch3CloseValueShow.lrValue	 := '        ;
aRecipeParamsVariables[384]:= 'stUCF.lrCapSorterPreScrewerBottleCatch4OpenValueShow.lrValue	 := '        ;
aRecipeParamsVariables[385]:= 'stUCF.lrCapSorterPreScrewerBottleCatch4CloseValueShow.lrValue	 := '        ;
aRecipeParamsVariables[386]:= 'stUCF.lrCapSorterPreScrewerBottleCatchToleranceValueShow.lrValue := '    ;
aRecipeParamsVariables[387]:= 'stUCF.lrCapSorterPreScrewerCatchAngleOpenSV.lrValue := '        ;
aRecipeParamsVariables[388]:= 'stUCF.lrCapSorterPreScrewerWaitInPlaceTimeShow.lrValue := '              ;
aRecipeParamsVariables[389]:= 'stUCF.bCapSorterPreScrewerCatchAngleOpenEnaShow.bValue := '              ;
aRecipeParamsVariables[390]:= 'stUCF.bCapSorterPreScrewerPoundedInCap.bValue := '              ;
aRecipeParamsVariables[391]:= 'stUCF.lrCapSorterBottleHightShow.lrValue		 := '              ;
aRecipeParamsVariables[392]:= 'stUCF.lrCapSorterBottleNeckHightShow.lrValue	 := '              ;
aRecipeParamsVariables[393]:= 'stUCF.lrCapSorterCapHightShow.lrValue			 := '              ;
aRecipeParamsVariables[394]:= 'stUCF.lrCapSorterCapNeckHightShow.lrValue		 := '              ;
aRecipeParamsVariables[395]:= 'stUCF.lrCapSorterSpare1.lrValue := '   ;
aRecipeParamsVariables[396]:= 'stUCF.lrCapSorterSpare2.lrValue := '   ;
aRecipeParamsVariables[397]:= 'stUCF.lrCapSorterSpare3.lrValue := '   ;
aRecipeParamsVariables[398]:= 'stUCF.lrCapSorterSpare4.lrValue := '   ;
aRecipeParamsVariables[399]:= 'stUCF.lrCapSorterSpare5.lrValue := '   ;
aRecipeParamsVariables[400]:= 'stUCF.lrCapSorterSpare6.lrValue := '   ;
aRecipeParamsVariables[401]:= 'stUCF.lrCapSorterSpare7.lrValue := '   ;
aRecipeParamsVariables[402]:= 'stUBF.iBottleSorterProductTypeShow.diValue := '                  ;
aRecipeParamsVariables[403]:= 'stUBF.uiBottleSorterIndexShow.udiValue		 := '                  ;
aRecipeParamsVariables[404]:= 'stUBF.bBottleSorterHopperTransporterEnableShow.bValue								 := '   ;
aRecipeParamsVariables[405]:= 'stUBF.iBottleSorterHopperConveyorRunningSpeedSVShow.diValue							 := '   ;
aRecipeParamsVariables[406]:= 'stUBF.iBottleSorterHopperConveyorEmptyingSpeedSVShow.diValue							 := '   ;
aRecipeParamsVariables[407]:= 'stUBF.iBottleSorterDistanceToFindElementOnTransferConveyorLimitRunningSVShow.diValue	 := '   ;
aRecipeParamsVariables[408]:= 'stUBF.iBottleSorterDistanceToFindElementOnTransferConveyorLimitEmptyingSVShow.diValue := '   ;
aRecipeParamsVariables[409]:= 'stUBF.bBottleSorterTransferTransporterEnableShow.bValue								 := '   ;
aRecipeParamsVariables[410]:= 'stUBF.iBottleSorterTransferConveyorRunningSpeedSVShow.diValue						 := '   ;
aRecipeParamsVariables[411]:= 'stUBF.iBottleSorterTransferConveyorEmptyingSpeedSVShow.diValue						 := '   ;
aRecipeParamsVariables[412]:= 'stUBF.iBottleSorterDistanceToFindElementOnSupplyConveyorDownstairsLimitSVShow.diValue := '   ;
aRecipeParamsVariables[413]:= 'stUBF.bBottleSorterSupplyTransporterEnableShow.bValue			 := '                      ;
aRecipeParamsVariables[414]:= 'stUBF.uiBottleSorterSupplyTransporterRunningSpeedSVShow.udiValue	 := '                      ;
aRecipeParamsVariables[415]:= 'stUBF.uiBottleSorterSupplyTransporterEmptingSpeedSVShow.udiValue	 := '                      ;
aRecipeParamsVariables[416]:= 'stUBF.lrBottleSorterModuloMoveOffsetSVShow.lrValue				 := '                      ;
aRecipeParamsVariables[417]:= 'stUBF.iBottleSorterSensorsCountFirstConditionSVShow.diValue	 := '                      ;
aRecipeParamsVariables[418]:= 'stUBF.iBottleSorterSupplyTimeFirstConditionSVShow.diValue		 := '                      ;
aRecipeParamsVariables[419]:= 'stUBF.iBottleSorterSensorsCountSecondConditionMinSVShow.diValue	 := '                      ;
aRecipeParamsVariables[420]:= 'stUBF.iBottleSorterSensorsCountSecondConditionMaxSVShow.diValue	 := '                      ;
aRecipeParamsVariables[421]:= 'stUBF.iBottleSorterSupplyTimeSecondConditionSVShow.diValue		 := '                      ;
aRecipeParamsVariables[422]:= 'stUBF.iBottleSorterSensorsCountThirdConditionSVShow.diValue	 := '                      ;
aRecipeParamsVariables[423]:= 'stUBF.iBottleSorterSupplyTimeThirdConditionSVShow.diValue		 := '                      ;
aRecipeParamsVariables[424]:= 'stUBF.bBottleSorterWeelEnableShow.bValue				 := '                      ;
aRecipeParamsVariables[425]:= 'stUBF.lrBottleSorterWheelSpeedSVShow.lrValue			 := '                      ;
aRecipeParamsVariables[426]:= 'stUBF.lrBottleSorterWheelEmptyingSpeedSVShow.lrValue	 := '                      ;
aRecipeParamsVariables[427]:= 'stUBF.bBottleSorterBrushEnableShow.bValue			 := '                      ;
aRecipeParamsVariables[428]:= 'stUBF.lrBottleSorterBrushHeightPositionSVShow.lrValue	 := '                      ;
aRecipeParamsVariables[429]:= 'stUBF.iBottleSorterBrushRunningSpeedSVShow.diValue	 := '                      ;
aRecipeParamsVariables[430]:= 'stUBF.iBottleSorterBrushEmptyingSpeedSVShow.diValue	 := '                      ;
aRecipeParamsVariables[431]:= 'stUBF.bBottleSorterRobotEnableShow.bValue	 := '                      ;
aRecipeParamsVariables[432]:= 'stUBF.nBottleSorterRobotRecipeId.diValue		 := '                      ;
aRecipeParamsVariables[433]:= 'stUBF.lrBottleSorterRemainingTimeToSuctionShow.lrValue := '                      ;
aRecipeParamsVariables[434]:= 'stUBF.lrBottleSorterSuckerSuctionTimeShow.lrValue		 := '                      ;
aRecipeParamsVariables[435]:= 'stUBF.lrBottleSorterRemainingTimeToRejectShow.lrValue  := '                      ;
aRecipeParamsVariables[436]:= 'stUBF.lrBottleSorterEjectorPulseShow.lrValue           := '                      ;
aRecipeParamsVariables[437]:= 'stUBF.lrBottleSorterZPickAboveTheBottleSVShow.lrValue	 := '                      ;
aRecipeParamsVariables[438]:= 'stUBF.lrBottleSorterZPickMoveSVShow.lrValue			 := '                      ;
aRecipeParamsVariables[439]:= 'stUBF.lrBottleSorterSafetyHeightSVShow.lrValue		 := '                      ;
aRecipeParamsVariables[440]:= 'stUBF.bBottleSorterRecieverEnableShow.bValue				 := '                      ;
aRecipeParamsVariables[441]:= 'stUBF.bBottleSorterRecieverSlot1EnableShow.bValue		 := '                      ;
aRecipeParamsVariables[442]:= 'stUBF.bBottleSorterRecieverSlot2EnableShow.bValue		 := '                      ;
aRecipeParamsVariables[443]:= 'stUBF.bBottleSorterRecieverSlot3EnableShow.bValue		 := '                      ;
aRecipeParamsVariables[444]:= 'stUBF.lrBottleSorterRecieverHeightPositionSVShow.lrValue := '                      ;
aRecipeParamsVariables[445]:= 'stUCF.lrCapSorterPreScrewerPickerSpeedWhenScrewerShow.lrValue :='				;
aRecipeParamsVariables[446]:= 'stUBL.bROPPCappingEnableShow.bValue						:=	 '      ;
aRecipeParamsVariables[447]:= 'stUBL.bROPPDragEnableShow.bValue	 					:=   '          ;
aRecipeParamsVariables[448]:= 'stUBL.bROPPFeederEnableShow.bValue						:=   '      ;                           
aRecipeParamsVariables[449]:= 'stUBL.bROPPSlowerEnableShow.bValue	 					:=   '      ;                           
aRecipeParamsVariables[450]:= 'stUBL.iROPPCapping1ToolShow.diValue 					:=   '              ;                       
aRecipeParamsVariables[451]:= 'stUBL.iROPPCappingTime2Show.diValue  					:=   '      ;                           
aRecipeParamsVariables[452]:= 'stUBL.iROPPCappingTimeShow.diValue  					:=   '          ;                       
aRecipeParamsVariables[453]:= 'stUBL.iROPPFeederTimeDelayOffShow.diValue 				:=   '             ;              
aRecipeParamsVariables[454]:= 'stUBL.iROPPFeederTimeDelayOnShow.diValue  				:=   '            ;               
aRecipeParamsVariables[455]:= 'stUBL.iROPPFeederTimeToEmptySleeveErrorShow.diValue	    :=   '       ;                           
aRecipeParamsVariables[456]:= 'stUBL.lrROPPCappingHeightPosSVShow.lrValue			    :=   '          ;                           
aRecipeParamsVariables[457]:= 'stUBL.lrROPPCappingVelocitySVShow.lrValue	 			:=   '       ;                           
aRecipeParamsVariables[458]:= 'stUBL.lrROPPDragAccelerationShow.lrValue	 			:=   '           ;                       
aRecipeParamsVariables[459]:= 'stUBL.lrROPPDragDecelerationShow.lrValue	 			:=   '              ;                       
aRecipeParamsVariables[460]:= 'stUBL.lrROPPDragVelocityShow.lrValue	 				:=   '          ;                       
aRecipeParamsVariables[461]:= 'stUBL.lrROPPFeederHeightPosSVShow.lrValue	 			:=   '      ;                           
aRecipeParamsVariables[462]:= 'stUBL.nROPPSlowerVelocitySVShow.udiValue				:=   '              ;
END_METHOD

METHOD METH_RecipeStuctToFileStruct : BOOL
VAR_INPUT
END_VAR

